VAR_GLOBAL CONSTANT
	MAX_DWORD	: DWORD := 4294967295;
	MAX_DWORD_2	: DWORD := -1;
	MAX_TIME	: TIME := TO_TIME(MAX_DWORD);
END_VAR

(* stored: Version 1.1.0.1, ProductVersion 3.1.4024.11
   GVL CONSTANTS: Id {0452a4dc-aaf2-46b0-870a-ec45447b5375} *)
